(*
SPDX-FileCopyrightText: © 2026 Oleksandr Tiutyk <trofimich@gmail.com>
SPDX-License-Identifier: MIT
License: https://opensource.org/license/mit
*)

{attribute 'no_explicit_call' := 'do not call this function block directly'} 
FUNCTION_BLOCK SetErrorAndContinueExceptionHandlingPolicy EXTENDS Object IMPLEMENTS IExceptionHandlingPolicy
VAR
	{attribute 'hide'} 
	_ClassName : STRING := __POUNAME();
END_VAR

{attribute 'monitoring' := 'call'}
PROPERTY ClassName : REFERENCE TO STRING
GET
ClassName REF= _ClassName;
END_GET
END_PROPERTY

METHOD HandleException : EXCEPTION_REACTION
VAR_INPUT
	exception : IReadOnlyException;
	handlingObject : IObject;
END_VAR
VAR_IN_OUT CONSTANT
	failedMethodName : STRING(255);
END_VAR
HandleException := EXCEPTION_REACTION.SET_ERROR_AND_CONTINUE;
END_METHOD

{attribute 'monitoring' := 'call'}
PROPERTY NamespaceName : REFERENCE TO STRING
GET
NamespaceName REF= CurrentNamespace.Name;
END_GET
END_PROPERTY

{attribute 'monitoring' := 'call'}
PROPERTY SelfSize : ULINT
GET
SelfSize := XSIZEOF(THIS^);
END_GET
END_PROPERTY

END_FUNCTION_BLOCK

(* stored: Version 1.1.0.1
   POU SetErrorAndContinueExceptionHandlingPolicy: Id {a4eb2320-3400-4dc2-8031-b55b6e1bbfa3}, SpecialFunc None
   Property ClassName: Id {3ac1fd6a-8981-46e7-88fa-adfce8200fbf}
   Get Get: Id {e0a59f69-f2b1-4954-bbc5-f99626dcbdee}
   Method HandleException: Id {462be713-1109-4737-a605-c6d09182fca9}
   Property NamespaceName: Id {12125e62-a5f3-4101-949a-c95b577951f5}
   Get Get: Id {d53a3505-556c-4128-a9b8-62085a2d05b4}
   Property SelfSize: Id {cd0a5ef3-cdc3-45f0-afdb-f57972fae1ca}
   Get Get: Id {9eb177ce-67e4-410e-aed0-e7613e6a2b75} *)
